PROGRAM P_Light_Test_CFC
VAR
	fbLight				:	FB_Light;
	bOn					:	BOOL;
	bOff				:	BOOL;
	bControlLevel		:	BOOL;
END_VAR

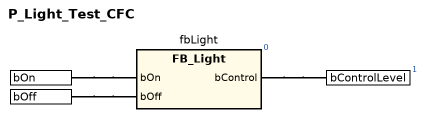
fbLight(bOn := bOn, bOff := bOff); // FB_Light
bControlLevel := fbLight.bControl;

END_PROGRAM

(* stored: Version 1.1.0.1, ProductVersion 3.1.4024.12
   POU P_Light_Test_CFC: Id {40eed654-30f9-4a77-ad89-5d5f035a4f47}, SpecialFunc None *)
